{attribute addProperty BoxType "EK1122-0000-0018"}
{attribute addProperty Id "Beckhoff_EL34xxsub_EK1100EK1100_179A0949162"}
{attribute addProperty CRC "1423978300"}
{attribute addProperty SizeInBites "16"}
{attribute addProperty SizeInBytes "2"}
TYPE Beckhoff_EL34xxEK1122_54E02F3C EXTENDS EK1122_179A0949 :
STRUCT
	{attribute addProperty Name "Beckhoff_EL34xxsub_EK1100"}
	Beckhoff_EL34xxsub_EK1100 : EK1100_179A0949;
END_STRUCT
END_TYPE

(* stored: Version 1.2.0.0, ProductVersion 3.1.4024.9
   DUT Beckhoff_EL34xxEK1122_54E02F3C: Id {82de2a18-3b39-4207-b82d-909a7691caf6} *)
